FUNCTION_BLOCK _TemplateTest EXTENDS TcUnit.FB_TestSuite
VAR
END_VAR

ExampleTest();

METHOD ExampleTest : BOOL
VAR
	expected : INT;
	actual : INT;
END_VAR
TcUnit.TEST('Example test');

expected := ;
actual := ;

AssertEquals(
	Expected := expected,
	Actual := actual,
	Message := 'What went wrong');

TEST_FINISHED();
END_METHOD

END_FUNCTION_BLOCK

(* stored: Version 1.1.0.1, ProductVersion 3.1.4024.12
   POU _TemplateTest: Id {046ee9eb-6990-07e4-3786-b4c9c68c548a}, SpecialFunc None
   Method ExampleTest: Id {43566aec-618b-0a5d-2cc8-6eea80d71980} *)
